// TIA Portal V18 export
// export: Created 2026-01-09T11:23:37.9996649Z, ExportSetting WithDefaults, DisplayName Totally Integrated Automation Portal, DisplayVersion V18 Update 5, DisplayName TIA Portal Openness, DisplayVersion V18 Update 5, DisplayName TIA Portal Teamcenter Gateway, DisplayVersion V18, DisplayName TIA Portal Version Control Interface, DisplayVersion V18, DisplayName SINAMICS Startdrive Advanced, DisplayVersion V18 SP2 Update 1, DisplayName SINAMICS Startdrive G110M, G120, G120C, G120D, G120P, G115D, DisplayVersion V18 SP2 Update 1, DisplayName SINAMICS Startdrive G130, G150, S120, S150, SINAMICS MV, S210, G220, S200, DisplayVersion V18 SP2 Update 1, DisplayName STEP 7 Professional, DisplayVersion V18 Update 5, DisplayName STEP 7 Safety, DisplayVersion V18, DisplayName WinCC Professional, DisplayVersion V18 Update 5
Screen "501 FixtureCheck"  1280x800, Number=501, Template=T1
  ScreenLayer 
    FaceplateInstance "FixtureCheck_2" at 0,180 size 1280x81  FaceplateTypeName=500 User@$@100 FixtureCheck@$@FixtureCheck_TP700 V 1.0.1
      InterfacePropertyText "FixtureName"  Text="工装2"
    FaceplateInstance "FixtureCheck_1" at 0,95 size 1280x81  FaceplateTypeName=500 User@$@100 FixtureCheck@$@FixtureCheck_TP700 V 1.0.1
      InterfacePropertyText "FixtureName"  Text="工装1"
    Button "btnMenu3" at 256,725 size 128x75  Mode=Text, StyleItem=BtnNormal20, TextOff="工装显示"
      on Press: ActivateScreen(Screen name := , Object number := 0)
